{attribute 'GeneratedUsingTerminal: EL1512-0000-0016'}
{attribute addProperty BoxType "EL1512-0000-0016"}
{attribute addProperty Id "CNT_Inputs_Channel_1AT %I*CNT_Inputs_Channel_21E1BB398CNT_Inputs_Channel_2AT %I*CNT_Inputs_Channel_21E1BB398CNT_Outputs_Channel_1AT %Q*CNT_Outputs_Channel_774A30BC6CNT_Outputs_Channel_2AT %Q*CNT_Outputs_Channel_774A30BC6WcStateAT %I*WcState_9091E0EB2InfoDataAT %I*InfoData_94A18F5E2"}
{attribute addProperty CRC "2339292382"}
{attribute addProperty Size "32"}
TYPE EL1512_8B6EC4DE EXTENDS EtcSlaveTerminalBase_947E5A46 :
STRUCT
	{attribute addProperty Name "CNT_Inputs_Channel_1"}
	CNT_Inputs_Channel_1 : CNT_Inputs_Channel_21E1BB39;
	{attribute addProperty Name "CNT_Inputs_Channel_2"}
	CNT_Inputs_Channel_2 : CNT_Inputs_Channel_21E1BB39;
	{attribute addProperty Name "CNT_Outputs_Channel_1"}
	CNT_Outputs_Channel_1 : CNT_Outputs_Channel_774A30BC;
	{attribute addProperty Name "CNT_Outputs_Channel_2"}
	CNT_Outputs_Channel_2 : CNT_Outputs_Channel_774A30BC;
	{attribute addProperty Name "WcState"}
	WcState : WcState_9091E0EB;
	{attribute addProperty Name "InfoData"}
	InfoData : InfoData_94A18F5E;
END_STRUCT
END_TYPE

(* stored: Version 1.2.0.0, ProductVersion 3.1.4024.9
   DUT EL1512_8B6EC4DE: Id {a9426a38-0263-42aa-b5fb-30a2a810f035} *)
